// TwinCAT 3 PLC project Untitled1
// ProgramVersion: 3.1.0.8
// libraries:
//   VisuElem3DPath, 3.5.4.0 (System)
//   VisuElemMeter, 3.5.4.0 (System)
//   VisuElems, 3.5.4.10 (System)
//   VisuElemsSpecialControls, 3.5.4.10 (System)
//   VisuElemsWinControls, 3.5.4.10 (System)
//   VisuElemTextEditor, 3.5.4.0 (System)
//   visuinputs, 3.5.4.0 (system)
//   VisuNativeControl, 3.5.4.0 (System)
//   Tc2_Standard, * (Beckhoff Automation GmbH)
//   Tc2_System, * (Beckhoff Automation GmbH)
//   Tc3_Interfaces, * (Beckhoff Automation GmbH)
//   Tc3_Module, * (Beckhoff Automation GmbH)
//   VisuDialogs, * (System)
//   Tc2_Utilities,3.3.7.0,Beckhoff Automation GmbH
// project tree:
//   DUTs/ E_PIZZA_TYPES.TcDUT, ST_PIZZA.TcDUT
//   / GlobalTextList.TcGTLO, PlcTask.TcTTO, Visualization Manager.TcVMO (not stored)
//   GVLs/ HMI_VARS.TcGVL
//   POUs/ MAIN.TcPOU, FB_PIZZA_OVEN.TcPOU, F_FIFO_WRITE.TcPOU
//   VISUs/ Visualization.TcVIS

CONFIGURATION Untitled1
    RESOURCE PLC ON TwinCAT3
        TASK PlcTask(INTERVAL := T#50000us, PRIORITY := 20);
        PROGRAM MAIN WITH PlcTask : MAIN;
    END_RESOURCE
END_CONFIGURATION

// ---- DUTs/E_PIZZA_TYPES.TcDUT
TYPE E_PIZZA_TYPES :
(
	eType_Cheese := 0,
	eType_Pepperoni := 1,
	eType_Sausage := 2
);
END_TYPE

// ---- DUTs/ST_PIZZA.TcDUT
TYPE ST_PIZZA :
STRUCT
	bExist : BOOL;
	dtTimeEnteredOven : DT;
	dtTimeExitedOven : DT;
	tTimeInOven : TIME;
	eType : E_PIZZA_TYPES; // 0 = Cheese, 1 = Pep, 2 = sausage
	
END_STRUCT
END_TYPE

// ---- GVLs/HMI_VARS.TcGVL
VAR_GLOBAL

	iState : DINT; // My machine state.
	bStartButton : BOOL;
	
	arrPizzaHistory : ARRAY [0..100] OF ST_PIZZA;
	
	fbNT_GetTime : NT_GetTime;
	stCurrentTime : TIMESTRUCT;
	dtCurrentTime : DT;
END_VAR

// ---- POUs/MAIN.TcPOU
PROGRAM MAIN
VAR

	fbMyPizzaOven : FB_PIZZA_OVEN;  // My Instance of oven 1
	
	bLoadPizza : BOOL;  // put a pizza on the input side
	bRemovePizza : BOOL;  // take pizza off output side.
	
	i : DINT;  
	
	arrMyBools : ARRAY [0..100] OF STRING;
	
	fbMyTimer : TON; 
	
END_VAR

VAR CONSTANT
	MAX_OVENS : DINT := 1; // This is 2.. 
END_VAR


fbMyPizzaOven(bLoadPizza:=bLoadPizza , bRemovePizza:=bRemovePizza );

fbMyTimer(IN:=NOT fbMyTimer.Q, PT:=T#100MS);

fbNT_GetTime(
	NETID:= '', 
	START:= fbMyTimer.Q , 
	TIMESTR=>hmi_vars.stCurrentTime );

END_PROGRAM

// ---- POUs/FB_PIZZA_OVEN.TcPOU
FUNCTION_BLOCK FB_PIZZA_OVEN
VAR_INPUT


	bLoadPizza : BOOL;  // put a pizza on the input side
	bRemovePizza : BOOL;  // take pizza off output side.

END_VAR
VAR_OUTPUT


	iTotalPizzasCooked : UDINT;			
	bBuzzer : BOOL;
	bLight : BOOL;  // NEW!

END_VAR
VAR

	fbLoad_RTRIG : R_TRIG;
	fbRemove_RTRIG : R_TRIG;

	iState : DINT;
	iLastState : DINT;
	sStateDesc : STRING;

	//timers
	fbMyTimer : TON;  // My Timer... for stuff.
	
	stPizzaOnDeck : ST_PIZZA; // Location of possible pizza... 
	stPizzaInOven : ST_PIZZA;  
	stPizzaDone   : ST_PIZZA; 
	
	arrStateDescHistory : ARRAY [1..100] OF STRING;

END_VAR
VAR CONSTANT
	stNULL_PIZZA : ST_PIZZA;  
END_VAR



dtCurrentTime := SYSTEMTIME_TO_DT(stCurrentTime);


// If there is room
IF stPizzaOnDeck.bExist AND NOT stPizzaInOven.bExist THEN
	stPizzaInOven := stPizzaOnDeck;
	stPizzaOnDeck := stNULL_PIZZA;  // Remove pizza.
END_IF


// Handle buttons... / sim inputs
fbLoad_RTRIG(clk := bLoadPizza);
IF fbLoad_RTRIG.Q THEN
	//bLoadPizza := FALSE;
	stPizzaOnDeck.bExist := TRUE;
	stPizzaOnDeck.eType := eType_Sausage;
END_IF

fbRemove_RTRIG(clk := bRemovePizza);
IF fbRemove_RTRIG.Q THEN
	F_FIFO_WRITE(cbData := SIZEOF(stPizzaDone), pData := ADR(stPizzaDone),
					cbBuffer := SIZEOF(arrPizzaHistory), pBuffer := ADR(arrPizzaHistory)
	);
	stPizzaDone := stNULL_PIZZA;
	//bRemovePizza := FALSE;
END_IF

CASE iState OF
	
	0:  // Wait for pizza in oven.
		sStateDesc := 'Waiting on Pizza Now.';
		IF stPizzaInOven.bExist THEN
			stPizzaInOven.dtTimeEnteredOven := dtCurrentTime;
			iState := 10;
		END_IF

	10: // We just got a pizza! Cook it.
		sStateDesc := 'Baking That Pizza Now.';
		fbMyTimer(IN:=TRUE,PT:=T#3S);
		IF fbMyTimer.Q THEN
			fbMyTimer(IN:=FALSE);
			iState := 20;	
		END_IF
 	
	
	20: // Can we move the pizza out of the oven?  Its going to burn.
	
		sStateDesc := 'PIZZA BURNING!!!!.';
	
		IF NOT stPizzaDone.bExist THEN
		
			//Simulate conveyor.
			stPizzaInOven.dtTimeExitedOven := dtCurrentTime;
			stPizzaDone := stPizzaInOven;
			stPizzaInOven := stNULL_PIZZA;
			bBuzzer := FALSE;
	
			iState := 30;
	
		ELSE
			
			bBuzzer := TRUE;
			
		END_IF
	
	30:  // Pizza just removed. on output tray.
	
		stPizzaDone.tTimeInOven := stPizzaDone.dtTimeExitedOven - stPizzaDone.dtTimeEnteredOven; 
		iTotalPizzasCooked := iTotalPizzasCooked + 1;
		iState := 0;   // Go wait for new pizza in oven!!

	
ELSE
	
	sStateDesc := 'Invalid state!';

END_CASE


// Start state history:

IF iLastState <> iState THEN

	// Do stuff here to log transitions.... 
	F_FIFO_WRITE(cbData := SIZEOF(sStateDesc), pData := ADR(sStateDesc),
					cbBuffer := SIZEOF(arrStateDescHistory), pBuffer := ADR(arrStateDescHistory)
	);
	
	// Reset for next time.
	iLastState := iState;

END_IF

END_FUNCTION_BLOCK

// ---- POUs/F_FIFO_WRITE.TcPOU
FUNCTION F_FIFO_WRITE : BOOL
VAR_INPUT
	cbData : UDINT;  // Stuff coming in.
	pData : POINTER TO BYTE;
	
	cbBuffer : UDINT;  // Where all the stuff lives.
	pBuffer : POINTER TO BYTE;
END_VAR
VAR
END_VAR



FW_MemMove(pDest := pBuffer + cbData, pSrc := pBuffer, cbLen := cbBuffer - cbData);


FW_MemMove(pDest := pBuffer, pSrc := pData, cbLen := cbData);

END_FUNCTION

// ---- GlobalTextList.TcGTLO
TEXTLIST GlobalTextList
  13 = 'B'
  7 = 'Buzzer'
  2 = 'Elapsed Tiime: %s'
  5 = 'Elapsed Time: '
  6 = 'Elapsed Time: %s'
  1 = 'Insert Pizza'
  3 = 'Insert Pizza '
  14 = 'L'
  8 = 'Light'
  12 = 'New Pizza Ready'
  11 = 'Package Pizza'
  0 = 'Pizza'
  10 = 'Pizza (Done)'
  9 = 'Pizza (On Deck)'
  16 = 'Pizzas Cooked %d'
  15 = 'Pizzas Cooked %I'
  17 = 'Pizzas Cooked: %d'
  18 = 'Status: %s'
  4 = 'Take Pizza Out'
END_TEXTLIST

// ---- VISUs/Visualization.TcVIS
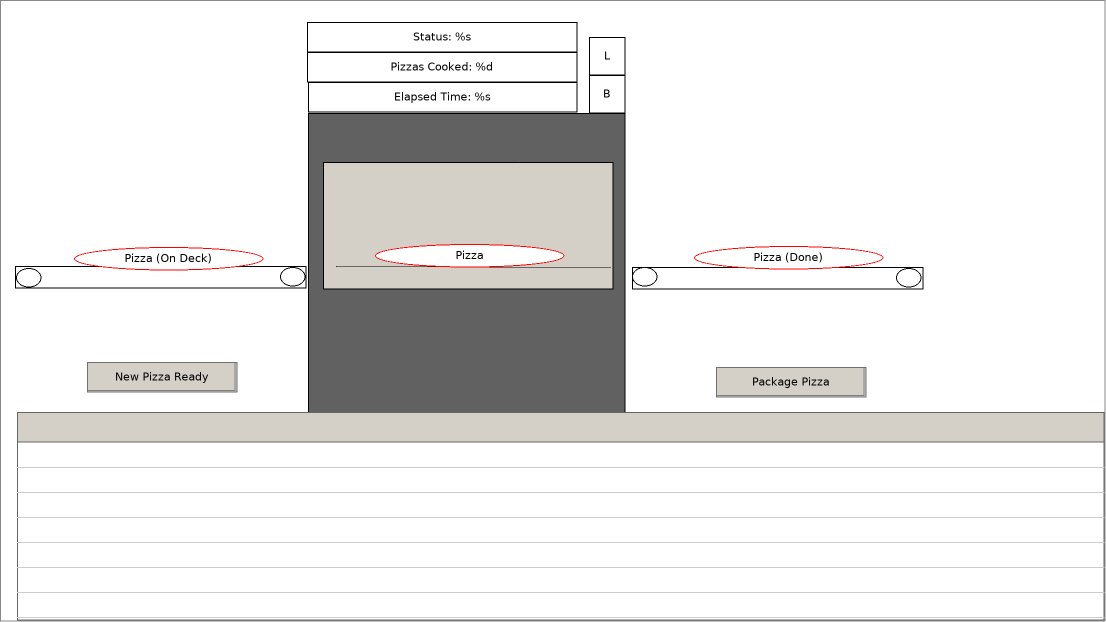
VISUALIZATION Visualization  // 1106x622
    Rectangle (308,113 317x477)
    Button (87,362 150x30), "New Pizza Ready"
        tap MAIN.bLoadPizza
    Button (716,367 150x30), "Package Pizza"
        tap MAIN.bRemovePizza
    Button (503,164 18x0)
    Rectangle (323,162 290x127)
    Rectangle (308,82 269x30), "Elapsed Time: %s", text variable: MAIN.fbMyPizzaOven.fbMyTimer.ET
    RoundedRectangle (15,266 291x22)
    RoundedRectangle (632,267 291x22)
    Ellipse (694,246 189x23), "Pizza (Done)", invisible if: NOT MAIN.fbMyPizzaOven.stPizzaDone.bExist
    Ellipse (74,247 189x23), "Pizza (On Deck)", invisible if: NOT MAIN.fbMyPizzaOven.stPizzaOnDeck.bExist
    Line (336,266) (610,267)
    Ellipse (375,244 189x23), "Pizza", invisible if: NOT MAIN.fbMyPizzaOven.stPizzaInOven.bExist
    RoundedRectangle (589,75 36x38), "B", colour toggle: MAIN.fbMyPizzaOven.bBuzzer
    RoundedRectangle (589,37 36x38), "L", colour toggle: MAIN.fbMyPizzaOven.bLight
    Rectangle (307,52 270x30), "Pizzas Cooked: %d", text variable: MAIN.fbMyPizzaOven.iTotalPizzasCooked
    Ellipse (16,268 25x19)
    Ellipse (280,267 25x19)
    Ellipse (632,267 25x19)
    Ellipse (896,268 25x19)
    Rectangle (307,22 270x30), "Status: %s", text variable: MAIN.fbMyPizzaOven.sStateDesc
    Table (17,412 1087x208), data array: HMI_VARS.arrPizzaHistory
        p3854506369: HMI_VARS.arrPizzaHistory[INDEX].bExist
        p1892666644: HMI_VARS.arrPizzaHistory[INDEX].dtTimeEnteredOven
        p338671338: HMI_VARS.arrPizzaHistory[INDEX].dtTimeExitedOven
        p2170511999: HMI_VARS.arrPizzaHistory[INDEX].tTimeInOven
        p3723444502: HMI_VARS.arrPizzaHistory[INDEX].eType
END_VISUALIZATION
